(* PLC project Generated.project, CODESYS CODESYS V3.5 SP19 Patch 1 *)
(* stored: creationDateTime 2026-08-23T01:36:48.751994, modificationDateTime 2026-08-23T01:36:48.751994 *)

(* values of E_Mode: DISABLE: Mode Désactivé / Veille de sécurité (sorties bloquées); MAINT_N1: Manuel Niveau 1 : Pilotage unitaire avec toutes sécurités actives; MAINT_N2: Manuel Niveau 2 : Pilotage dégradé (droits étendus + bypasses autorisés); SEMI_AUTO: Mode Semi-Automatique (séquenceur automatique) *)

{attribute 'qualified_only'}
{attribute 'strict'}
TYPE E_Mode : (DISABLE := 0, MAINT_N1 := 1, MAINT_N2 := 2, SEMI_AUTO := 3);
END_TYPE

(* ======================================================================= 🧩 ST_FbStatus — Socle transverse de statut d'un FB métier ─────────────────────────────────────────────────────────────── 🎯 Rôle : regroupe l'état, le défaut et le warning d'un FB standard, avec les textes prêts pour l'IHM (plus de conditions complexes côté affichage). Évolution additive : les 6 membres d'origine sont conservés. 🧬 Forme cible : les FB standard exposent `Status : ST_FbStatus` rempli via le socle `FB_FbStatus` (même comportement partout). ⚠️ State/StateAtError : E_State (phases opérationnelles FB métier). Un FB dont l'état est un énum domaine (E_Diag_State, CycleStep, ST_Safety_Emergency_State…) garde sa sortie typée SÉPARÉE et ne migre pas vers ST_FbStatus (exception documentée). 📄 Doc : DOC/STDS/CODE_QUALITY_STANDARDS.md §2quinquies ======================================================================= *)
TYPE ST_FbStatus : STRUCT
  Busy : BOOL;  (* ---- membres historiques (conservés) ---- 1 = Bloc en cours d'exécution *)
  Done : BOOL;  (* 1 = Action terminée avec succès *)
  Error : BOOL;  (* 1 = Défaut à acquitter (laté jusqu'au Reset) *)
  ErrorId : WORD;  (* Code d'erreur bitfield / enum diagnostic *)
  State : E_State;  (* État courant de la machine d'état *)
  StateAtError : E_State;  (* État mémorisé lors de l'apparition du défaut *)
  Warning : BOOL;  (* ---- membres ajoutés (forme cible enrichie) ---- 1 = warning actif (auto-effacé, aucun acquittement) *)
  WarningId : WORD;  (* Code warning courant (bitfield) *)
  WarningIdTxt : STRING;  (* Texte généré depuis WarningId (prêt IHM) *)
  ErrorIdTxt : STRING;  (* Texte généré depuis ErrorId *)
  ResetRequested : BOOL;  (* 1 = un Reset est nécessaire / en cours *)
END_STRUCT;
END_TYPE

(* values of E_State: DISABLED: Enable faux, neutralisé; INIT: Démarrage / vérifs; READY: Prêt, attend ordre; BUSY: Action en cours; DONE: Action terminée; STOPPING: Décél rampe avant arrêt (StartStop=FALSE ou SafeStop=TRUE) *)

{attribute 'qualified_only'}
{attribute 'strict'}
TYPE E_State : (DISABLED := 0, INIT := 1, READY := 2, BUSY := 3, DONE := 4, STOPPING := 5);
END_TYPE

(* ======================================================================= 📊 FB_Encoder_SpeedMonitor — Détection variation brusque vitesse câble ─────────────────────────────────────────────────────────────── 🎯 Rôle : Surveillance et détection de variation brusque de vitesse câble 🔒 Polarité : SpeedVariationConfirmed=TRUE si variation > seuil pendant timeout 📊 Diagnostic : Brique de surveillance diagnostic sans actionneur direct 📄 Doc métier : DOC/AF/AF_Partie-09_Fonction_Encoder_v2.1.md ======================================================================= *)
FUNCTION_BLOCK FB_Encoder_SpeedMonitor
  VAR_INPUT
    Enable : BOOL;  (* === COMMANDES & AUTORISATIONS === --> [CMD] Autorisation generale FB (TRUE=Autorise) *)
    Reset : BOOL;  (* --> [CMD] Acquittement defaut (front montant) *)
    PowerContactorEngaged : BOOL;  (* === CONTEXTE & ETAT PUISSANCE === --> [HW] Ligne puissance enclenchee *)
    Mode : E_Mode;  (* --> [CMD] Mode d'exploitation actif *)
    SpeedMps : REAL;  (* === MESURES & CONSIGNES SURVEILLANCE === --> [HW] Vitesse lineaire absolue mesuree (m/s) *)
    SpeedVariationThresholdMps : REAL;  (* --> [CFG] Seuil de variation minimale a surveiller (m/s) *)
    SpeedVariationTimeout : TIME;  (* --> [CFG] Duree minimale de confirmation variation *)
    SpeedStabilityTimeout : TIME;  (* --> [CFG] Duree sans variation avant vitesse stable *)
  END_VAR
  VAR_OUTPUT
    Ready : BOOL;  (* === ETATS IEC & SYNOPTIQUE === <-- [STAT] FB pret a fonctionner *)
    Status : ST_FbStatus;  (* 🧩 Statut transverse (forme cible) — regroupe Busy/Done/Error/ErrorId/State/StateAtError. ErrorId bit0: "variation vitesse confirmée". *)
    SpeedDeltaMps : REAL;  (* === RESULTATS & MESURES DIAGNOSTIC === <-- [DIAG] Ecart absolu entre deux mesures (m/s) *)
    SpeedVariationDetected : BOOL;  (* <-- [DIAG] Seuil depasse sur le cycle courant *)
    SpeedVariationConfirmed : BOOL;  (* <-- [DIAG] Seuil depasse pendant la duree requise *)
    SpeedStable : BOOL;  (* <-- [STAT] Vitesse stable pendant SpeedStabilityTimeout *)
  END_VAR
  VAR
    ResetEdge : R_TRIG;  (* === DETECTEURS DE FRONT === . [LOC] Detecteur front montant Reset *)
    ErrorEdge : R_TRIG;  (* . [LOC] Detecteur front montant Error *)
    VariationTimer : TON;  (* === TEMPORISATEURS INTERNES === . [LOC] Temporisateur de confirmation de variation *)
    StabilityTimer : TON;  (* . [LOC] Temporisateur de confirmation de stabilite *)
    PreviousSpeedMps : REAL;  (* === VARIABLES ET MEMOIRES INTERNES === . [LOC] Vitesse mesuree au cycle precedent (m/s) *)
    HasPreviousSpeed : BOOL;  (* . [LOC] Premiere mesure enregistree *)
    VariationActive : BOOL;  (* . [LOC] Condition de depassement de seuil active *)
  END_VAR

            

{region "§1 Gate"}
// 🛑 1. GATE — désactivation ou AU non réarmé : aucune alarme persistante.
IF NOT Enable OR NOT PowerContactorEngaged THEN
    Ready := FALSE;
    Status.Busy := FALSE;
    Status.Done := FALSE;
    Status.Error := FALSE;
    Status.ErrorId := 16#0000;
    Status.State := E_State.DISABLED;
    SpeedDeltaMps := 0.0;
    SpeedVariationDetected := FALSE;
    SpeedVariationConfirmed := FALSE;
    SpeedStable := FALSE;
    VariationActive := FALSE;
    HasPreviousSpeed := FALSE;
    VariationTimer(IN := FALSE, PT := SpeedVariationTimeout);
    StabilityTimer(IN := FALSE, PT := SpeedStabilityTimeout);
    RETURN;
END_IF;

Ready := TRUE;
Status.Busy := FALSE;
Status.Done := FALSE;
Status.State := E_State.READY;
{endregion}

{region "§2 Reset front"}
// 🔑 2. RESET FRONT — l'acquittement n'efface le défaut que si la cause a disparu.
ResetEdge(CLK := Reset);
{endregion}

{region "§3 Calcul écart vitesse"}
// 📏 3. CALCUL DE L'ÉCART DE VITESSE — première mesure utilisée comme référence.
IF NOT HasPreviousSpeed THEN
    PreviousSpeedMps := SpeedMps;
    HasPreviousSpeed := TRUE;
    SpeedDeltaMps := 0.0;
ELSE
    SpeedDeltaMps := ABS(SpeedMps - PreviousSpeedMps);
    PreviousSpeedMps := SpeedMps;
END_IF;
{endregion}

{region "§4 Détection et filtre temporel"}
// 🔍 4. DÉTECTION BRUTE + FILTRE TEMPOREL — pas de déclenchement si la durée vaut zéro.
VariationActive := HasPreviousSpeed
                   AND (SpeedVariationThresholdMps >= 0.0)
                   AND (SpeedVariationTimeout > T#0ms)
                   AND (SpeedDeltaMps > SpeedVariationThresholdMps);
SpeedVariationDetected := VariationActive;

VariationTimer(IN := VariationActive, PT := SpeedVariationTimeout);
SpeedVariationConfirmed := VariationTimer.Q;
StabilityTimer(IN := HasPreviousSpeed AND NOT VariationActive AND (SpeedStabilityTimeout > T#0ms), PT := SpeedStabilityTimeout);
SpeedStable := StabilityTimer.Q;

IF SpeedVariationConfirmed THEN
    Status.ErrorId := Status.ErrorId OR 16#0001;
ELSIF ResetEdge.Q AND NOT VariationActive THEN
    Status.ErrorId := Status.ErrorId AND 16#FFFE;
END_IF;
{endregion}

{region "§5 Sorties état"}
// 📤 5. SORTIES D'ÉTAT — diagnostic standard, aucune commande mouvement.
Status.Error := (Status.ErrorId <> 16#0000);
ErrorEdge(CLK := Status.Error);
IF ErrorEdge.Q THEN
    Status.StateAtError := Status.State;
END_IF;
{endregion}

          
END_FUNCTION_BLOCK
